PROGRAM PRG_PAOL_01_LightboxScanersCtrl
VAR

	tonEnableCameraSystem					: TON;
	bEnablePackAggregationCameraSystem		: BOOL;
	bEnablePackTriggeringAfterDelayON		: BOOL;

	tofPackAggregationCameraOFFDelay 		: TOF;
	bEnablePackTriggeringAfterDelayOFF		: BOOL;

	fbPuls							: FB_Puls;
	tonLightboxLensAirNextBlow		: TON;
	//rtLightboxLensAirBlowing		: R_TRIG;
	tonLightboxLensAirBlowing		: TOF;

	fbCameraBoxRead					: FB_2CAM_CameraBoxRead;
	aScannerCtrl					: ARRAY[1..2] OF FB_SCANNER_CameraSelect;
	aCodeDiag						: ARRAY[1..2] OF FB_SCANNER_DiagnosticLog;

	bCameraTriggersArmed			: BOOL;
	bCameraTrigger1Conditioned		: BOOL;
	bCameraTrigger2Conditioned		: BOOL;
	bCameraTrigger3Conditioned		: BOOL;
	bCameraTrigger4Conditioned		: BOOL;
	bCameraTrigger5Conditioned		: BOOL;
	bCameraTrigger6Conditioned		: BOOL;

	rtCameraTrigger					: ARRAY[0..6] OF R_TRIG;
	aCameraTrigger					: ARRAY[0..6] OF BOOL;

	fbCameraSequenceNo				: FB_2CAM_CameraSequenceNo;

	fbPackScanners_2x5Packs			: FB_2CAM_PackScanners2x5Packs;
	fbSelectCameraMap				: FB_2CAM_SelectCameraMap;

	fbAddNewOuterTriggerID			: FB_PAOL_AddNewTriggerID;
	fbMoveOuterStatusArray			: FB_PACK_MoveOuterStatusArray;	(*Actually is moving OCVPackStatusArray*)

	aAddPackCodes					: ARRAY[1..2] OF FB_2CAM_AddPackCodes;
	aPackScanner					: ARRAY[1..2] OF ST_SCANNER_CameraMap;
	aPackCameraEvaluation			: ARRAY[1..2] OF FB_SCANNER_Evaluation;

	bPackCodeDataInvalid			: BOOL;
	ctuConsecutiveDataInvalid		: CTU;

	aInfeedCamerasSync 				: ARRAY[1..2] OF FB_PAOL_InfeedCamerasSync;

	tonDelayStopOuter				: TON;


END_VAR
VAR // added by the converter: edge detectors and wires of the graphical bodies
    _w1, _w3 : BOOL;
    _w2 : UDINT;
END_VAR

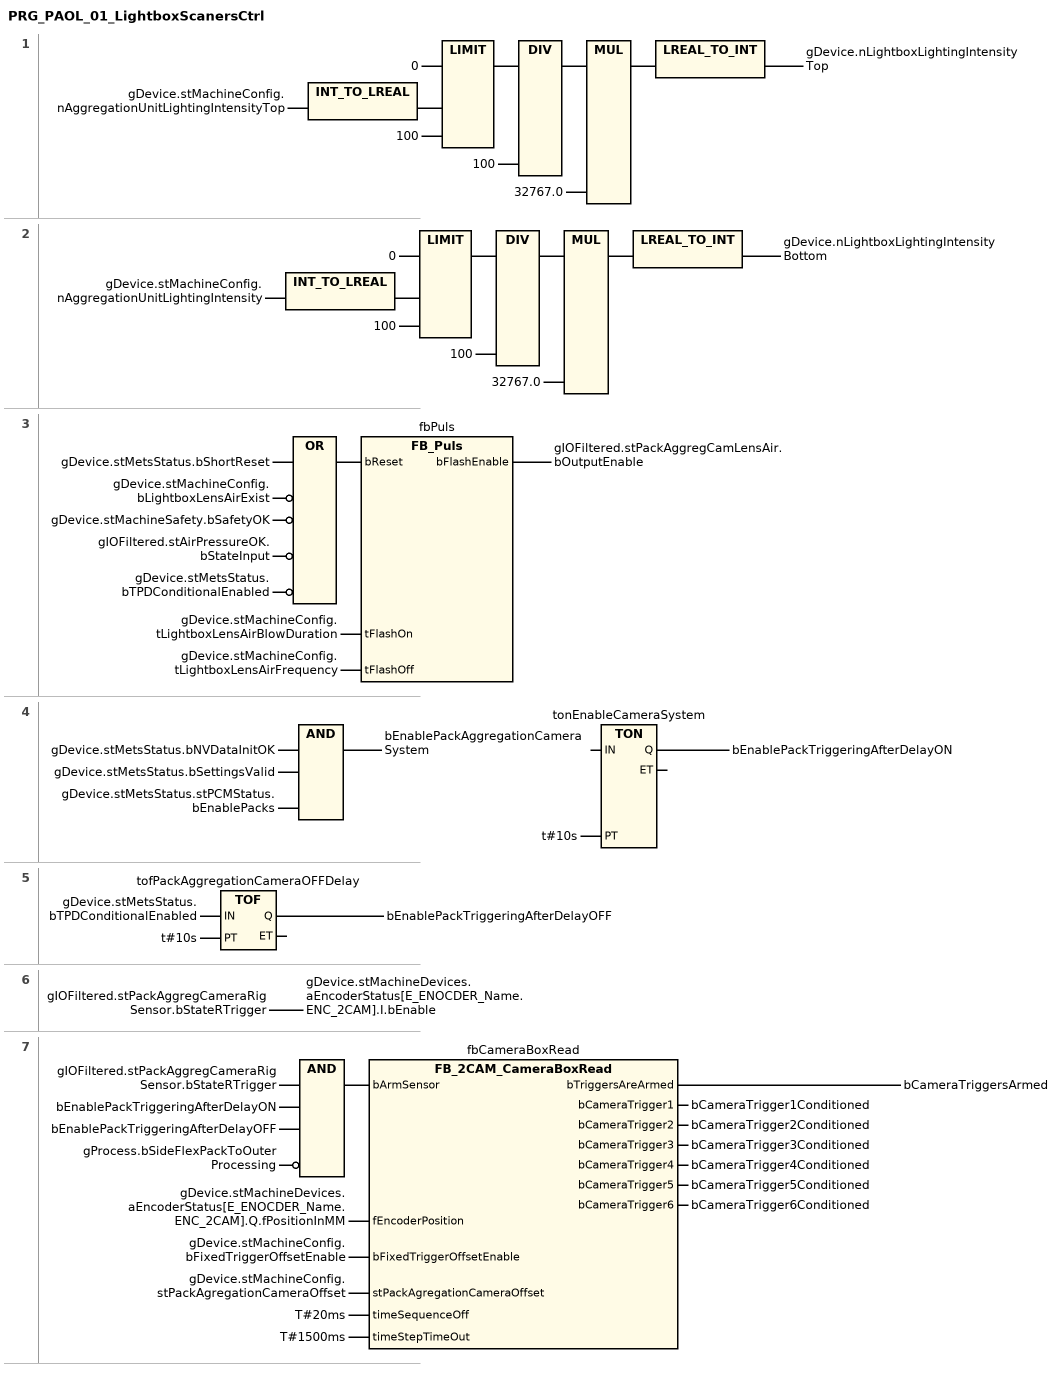
// NETWORK 1
gDevice.nLightboxLightingIntensityTop := LREAL_TO_INT((LIMIT(0, INT_TO_LREAL(gDevice.stMachineConfig.nAggregationUnitLightingIntensityTop), 100) / 100) * 32767.0);

// NETWORK 2
gDevice.nLightboxLightingIntensityBottom := LREAL_TO_INT((LIMIT(0, INT_TO_LREAL(gDevice.stMachineConfig.nAggregationUnitLightingIntensity), 100) / 100) * 32767.0);

// NETWORK 3
fbPuls(
    bReset := gDevice.stMetsStatus.bShortReset OR NOT gDevice.stMachineConfig.bLightboxLensAirExist OR NOT gDevice.stMachineSafety.bSafetyOK OR NOT gIOFiltered.stAirPressureOK.bStateInput OR NOT gDevice.stMetsStatus.bTPDConditionalEnabled,
    tFlashOn := gDevice.stMachineConfig.tLightboxLensAirBlowDuration,
    tFlashOff := gDevice.stMachineConfig.tLightboxLensAirFrequency); // FB_Puls
gIOFiltered.stPackAggregCamLensAir.bOutputEnable := fbPuls.bFlashEnable;

// NETWORK 4
_w1 := gDevice.stMetsStatus.bNVDataInitOK AND gDevice.stMetsStatus.bSettingsValid AND gDevice.stMetsStatus.stPCMStatus.bEnablePacks;
bEnablePackAggregationCameraSystem := _w1;
tonEnableCameraSystem(IN := _w1, PT := t#10s); // TON
bEnablePackTriggeringAfterDelayON := tonEnableCameraSystem.Q;

// NETWORK 5
tofPackAggregationCameraOFFDelay(IN := gDevice.stMetsStatus.bTPDConditionalEnabled, PT := t#10s); // TOF
bEnablePackTriggeringAfterDelayOFF := tofPackAggregationCameraOFFDelay.Q;

// NETWORK 6
gDevice.stMachineDevices.aEncoderStatus[E_ENOCDER_Name.ENC_2CAM].I.bEnable := gIOFiltered.stPackAggregCameraRigSensor.bStateRTrigger;

// NETWORK 7
fbCameraBoxRead(
    bArmSensor := gIOFiltered.stPackAggregCameraRigSensor.bStateRTrigger AND bEnablePackTriggeringAfterDelayON AND bEnablePackTriggeringAfterDelayOFF AND NOT gProcess.bSideFlexPackToOuterProcessing,
    fEncoderPosition := gDevice.stMachineDevices.aEncoderStatus[E_ENOCDER_Name.ENC_2CAM].Q.fPositionInMM,
    bFixedTriggerOffsetEnable := gDevice.stMachineConfig.bFixedTriggerOffsetEnable,
    stPackAgregationCameraOffset := gDevice.stMachineConfig.stPackAgregationCameraOffset,
    timeSequenceOff := T#20ms,
    timeStepTimeOut := T#1500ms,
    bCameraTrigger1 => bCameraTrigger1Conditioned,
    bCameraTrigger2 => bCameraTrigger2Conditioned,
    bCameraTrigger3 => bCameraTrigger3Conditioned,
    bCameraTrigger4 => bCameraTrigger4Conditioned,
    bCameraTrigger5 => bCameraTrigger5Conditioned,
    bCameraTrigger6 => bCameraTrigger6Conditioned); // FB_2CAM_CameraBoxRead
bCameraTriggersArmed := fbCameraBoxRead.bTriggersAreArmed;

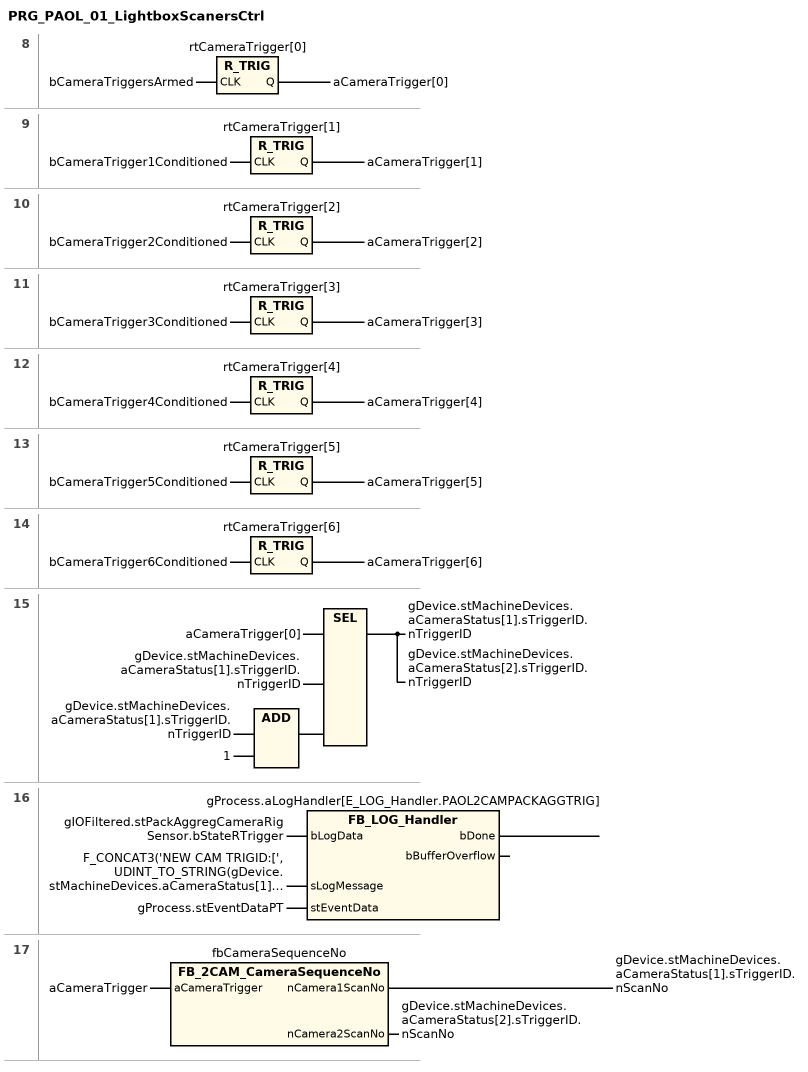
// NETWORK 8
rtCameraTrigger[0](CLK := bCameraTriggersArmed); // R_TRIG
aCameraTrigger[0] := rtCameraTrigger[0].Q;

// NETWORK 9
rtCameraTrigger[1](CLK := bCameraTrigger1Conditioned); // R_TRIG
aCameraTrigger[1] := rtCameraTrigger[1].Q;

// NETWORK 10
rtCameraTrigger[2](CLK := bCameraTrigger2Conditioned); // R_TRIG
aCameraTrigger[2] := rtCameraTrigger[2].Q;

// NETWORK 11
rtCameraTrigger[3](CLK := bCameraTrigger3Conditioned); // R_TRIG
aCameraTrigger[3] := rtCameraTrigger[3].Q;

// NETWORK 12
rtCameraTrigger[4](CLK := bCameraTrigger4Conditioned); // R_TRIG
aCameraTrigger[4] := rtCameraTrigger[4].Q;

// NETWORK 13
rtCameraTrigger[5](CLK := bCameraTrigger5Conditioned); // R_TRIG
aCameraTrigger[5] := rtCameraTrigger[5].Q;

// NETWORK 14
rtCameraTrigger[6](CLK := bCameraTrigger6Conditioned); // R_TRIG
aCameraTrigger[6] := rtCameraTrigger[6].Q;

// NETWORK 15
_w2 := SEL(aCameraTrigger[0], gDevice.stMachineDevices.aCameraStatus[1].sTriggerID.nTriggerID, gDevice.stMachineDevices.aCameraStatus[1].sTriggerID.nTriggerID + 1);
gDevice.stMachineDevices.aCameraStatus[1].sTriggerID.nTriggerID := _w2;
gDevice.stMachineDevices.aCameraStatus[2].sTriggerID.nTriggerID := _w2;

// NETWORK 16
gProcess.aLogHandler[E_LOG_Handler.PAOL2CAMPACKAGGTRIG](
    bLogData := gIOFiltered.stPackAggregCameraRigSensor.bStateRTrigger,
    sLogMessage := F_CONCAT3('NEW CAM TRIGID:[', UDINT_TO_STRING(gDevice.stMachineDevices.aCameraStatus[1].sTriggerID.nTriggerID), ']'),
    stEventData := gProcess.stEventDataPT); // FB_LOG_Handler

// NETWORK 17
fbCameraSequenceNo(aCameraTrigger := aCameraTrigger, nCamera2ScanNo => gDevice.stMachineDevices.aCameraStatus[2].sTriggerID.nScanNo); // FB_2CAM_CameraSequenceNo
gDevice.stMachineDevices.aCameraStatus[1].sTriggerID.nScanNo := fbCameraSequenceNo.nCamera1ScanNo;

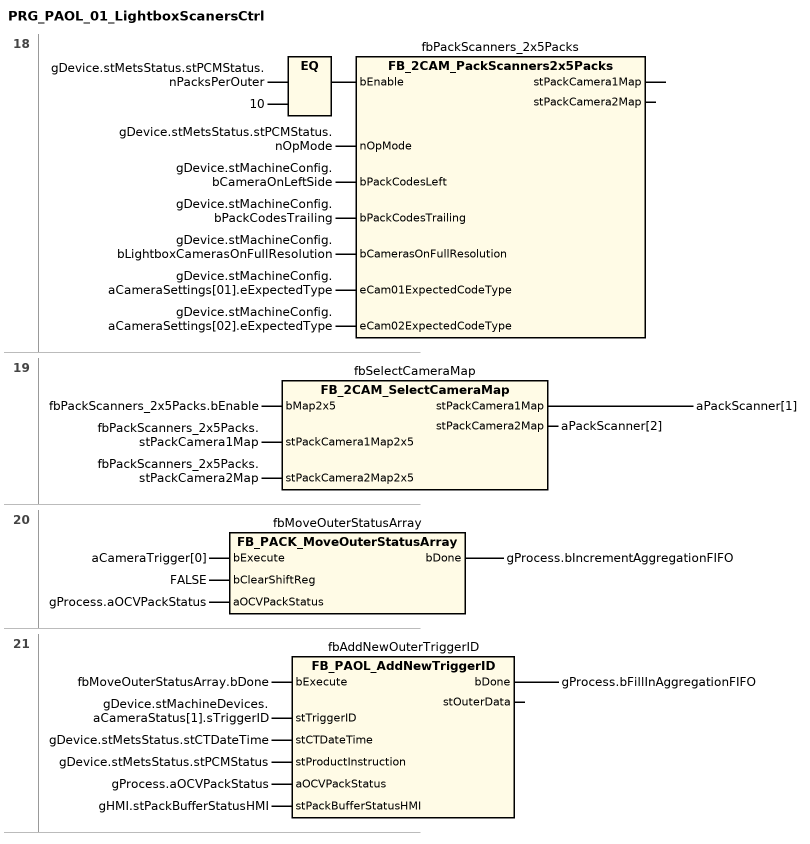
// NETWORK 18
fbPackScanners_2x5Packs(
    bEnable := gDevice.stMetsStatus.stPCMStatus.nPacksPerOuter = 10,
    nOpMode := gDevice.stMetsStatus.stPCMStatus.nOpMode,
    bPackCodesLeft := gDevice.stMachineConfig.bCameraOnLeftSide,
    bPackCodesTrailing := gDevice.stMachineConfig.bPackCodesTrailing,
    bCamerasOnFullResolution := gDevice.stMachineConfig.bLightboxCamerasOnFullResolution,
    eCam01ExpectedCodeType := gDevice.stMachineConfig.aCameraSettings[01].eExpectedType,
    eCam02ExpectedCodeType := gDevice.stMachineConfig.aCameraSettings[02].eExpectedType); // FB_2CAM_PackScanners2x5Packs

// NETWORK 19
fbSelectCameraMap(
    bMap2x5 := fbPackScanners_2x5Packs.bEnable,
    stPackCamera1Map2x5 := fbPackScanners_2x5Packs.stPackCamera1Map,
    stPackCamera2Map2x5 := fbPackScanners_2x5Packs.stPackCamera2Map,
    stPackCamera2Map => aPackScanner[2]); // FB_2CAM_SelectCameraMap
aPackScanner[1] := fbSelectCameraMap.stPackCamera1Map;

// NETWORK 20
fbMoveOuterStatusArray(
    bExecute := aCameraTrigger[0],
    bClearShiftReg := FALSE,
    aOCVPackStatus := gProcess.aOCVPackStatus); // FB_PACK_MoveOuterStatusArray
gProcess.bIncrementAggregationFIFO := fbMoveOuterStatusArray.bDone;

// NETWORK 21
fbAddNewOuterTriggerID(
    bExecute := fbMoveOuterStatusArray.bDone,
    stTriggerID := gDevice.stMachineDevices.aCameraStatus[1].sTriggerID,
    stCTDateTime := gDevice.stMetsStatus.stCTDateTime,
    stProductInstruction := gDevice.stMetsStatus.stPCMStatus,
    aOCVPackStatus := gProcess.aOCVPackStatus,
    stPackBufferStatusHMI := gHMI.stPackBufferStatusHMI); // FB_PAOL_AddNewTriggerID
gProcess.bFillInAggregationFIFO := fbAddNewOuterTriggerID.bDone;

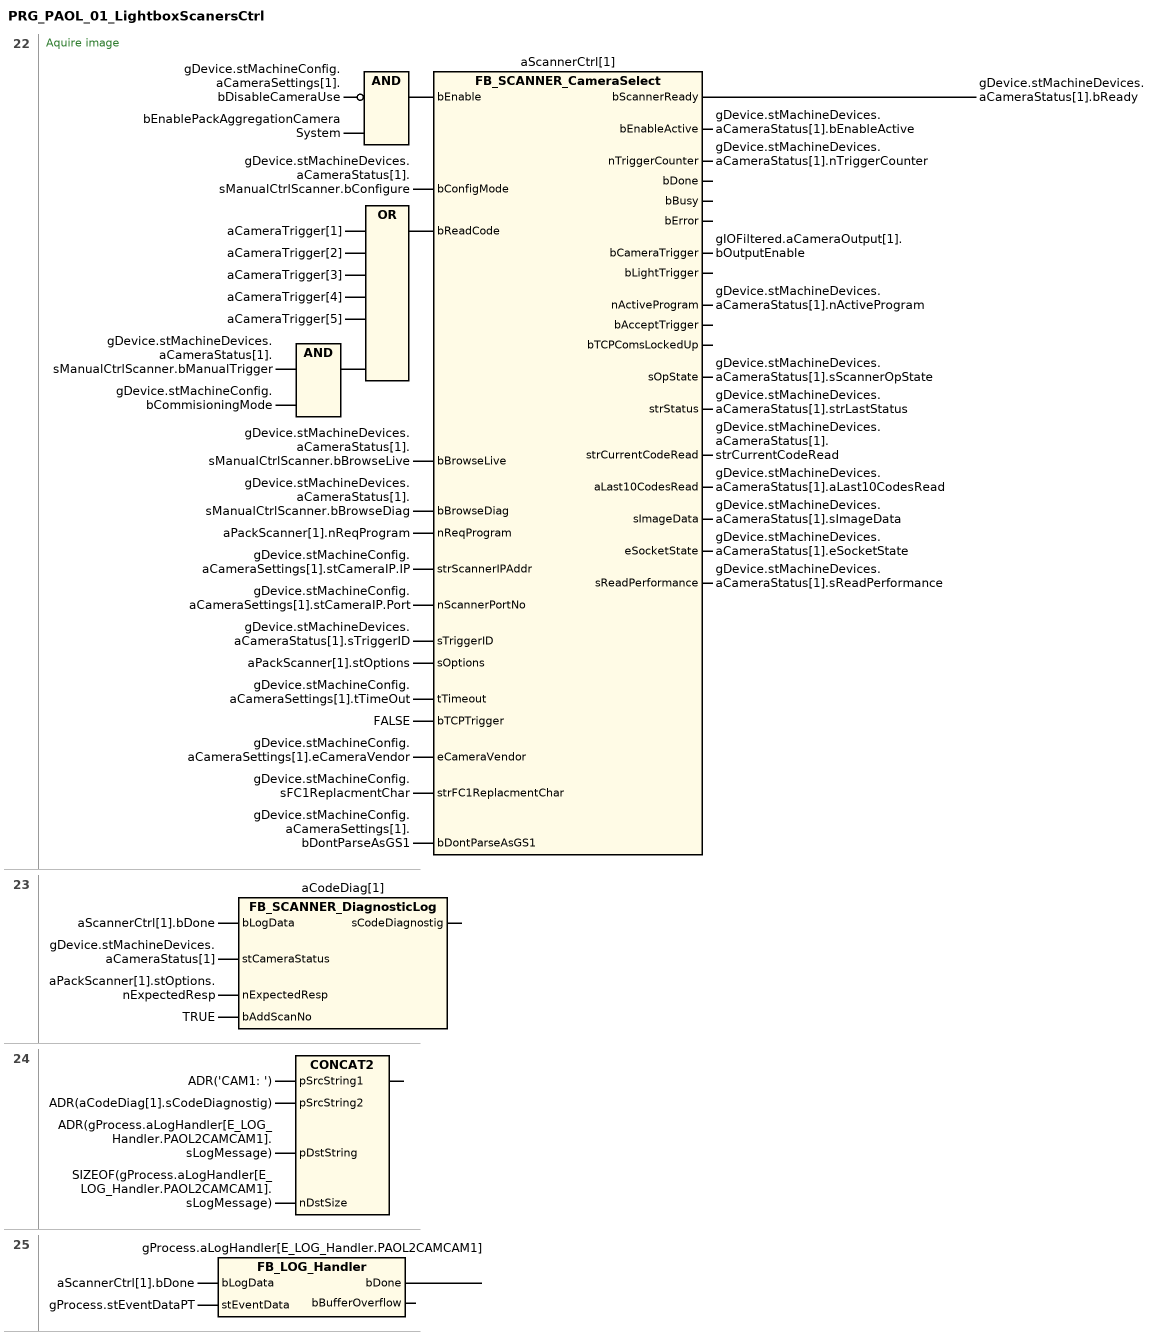
// NETWORK 22
// Aquire image
aScannerCtrl[1](
    bEnable := NOT gDevice.stMachineConfig.aCameraSettings[1].bDisableCameraUse AND bEnablePackAggregationCameraSystem,
    bConfigMode := gDevice.stMachineDevices.aCameraStatus[1].sManualCtrlScanner.bConfigure,
    bReadCode := aCameraTrigger[1] OR aCameraTrigger[2] OR aCameraTrigger[3] OR aCameraTrigger[4] OR aCameraTrigger[5] OR gDevice.stMachineDevices.aCameraStatus[1].sManualCtrlScanner.bManualTrigger AND gDevice.stMachineConfig.bCommisioningMode,
    bBrowseLive := gDevice.stMachineDevices.aCameraStatus[1].sManualCtrlScanner.bBrowseLive,
    bBrowseDiag := gDevice.stMachineDevices.aCameraStatus[1].sManualCtrlScanner.bBrowseDiag,
    nReqProgram := aPackScanner[1].nReqProgram,
    strScannerIPAddr := gDevice.stMachineConfig.aCameraSettings[1].stCameraIP.IP,
    nScannerPortNo := gDevice.stMachineConfig.aCameraSettings[1].stCameraIP.Port,
    sTriggerID := gDevice.stMachineDevices.aCameraStatus[1].sTriggerID,
    sOptions := aPackScanner[1].stOptions,
    tTimeout := gDevice.stMachineConfig.aCameraSettings[1].tTimeOut,
    bTCPTrigger := FALSE,
    eCameraVendor := gDevice.stMachineConfig.aCameraSettings[1].eCameraVendor,
    strFC1ReplacmentChar := gDevice.stMachineConfig.sFC1ReplacmentChar,
    bDontParseAsGS1 := gDevice.stMachineConfig.aCameraSettings[1].bDontParseAsGS1,
    bEnableActive => gDevice.stMachineDevices.aCameraStatus[1].bEnableActive,
    nTriggerCounter => gDevice.stMachineDevices.aCameraStatus[1].nTriggerCounter,
    bCameraTrigger => gIOFiltered.aCameraOutput[1].bOutputEnable,
    nActiveProgram => gDevice.stMachineDevices.aCameraStatus[1].nActiveProgram,
    sOpState => gDevice.stMachineDevices.aCameraStatus[1].sScannerOpState,
    strStatus => gDevice.stMachineDevices.aCameraStatus[1].strLastStatus,
    strCurrentCodeRead => gDevice.stMachineDevices.aCameraStatus[1].strCurrentCodeRead,
    aLast10CodesRead => gDevice.stMachineDevices.aCameraStatus[1].aLast10CodesRead,
    sImageData => gDevice.stMachineDevices.aCameraStatus[1].sImageData,
    eSocketState => gDevice.stMachineDevices.aCameraStatus[1].eSocketState,
    sReadPerformance => gDevice.stMachineDevices.aCameraStatus[1].sReadPerformance); // FB_SCANNER_CameraSelect
gDevice.stMachineDevices.aCameraStatus[1].bReady := aScannerCtrl[1].bScannerReady;

// NETWORK 23
aCodeDiag[1](
    bLogData := aScannerCtrl[1].bDone,
    stCameraStatus := gDevice.stMachineDevices.aCameraStatus[1],
    nExpectedResp := aPackScanner[1].stOptions.nExpectedResp,
    bAddScanNo := TRUE); // FB_SCANNER_DiagnosticLog

// NETWORK 24
CONCAT2(pSrcString1 := ADR('CAM1: '), pSrcString2 := ADR(aCodeDiag[1].sCodeDiagnostig), pDstString := ADR(gProcess.aLogHandler[E_LOG_Handler.PAOL2CAMCAM1].sLogMessage), nDstSize := SIZEOF(gProcess.aLogHandler[E_LOG_Handler.PAOL2CAMCAM1].sLogMessage));

// NETWORK 25
gProcess.aLogHandler[E_LOG_Handler.PAOL2CAMCAM1](bLogData := aScannerCtrl[1].bDone, stEventData := gProcess.stEventDataPT); // FB_LOG_Handler

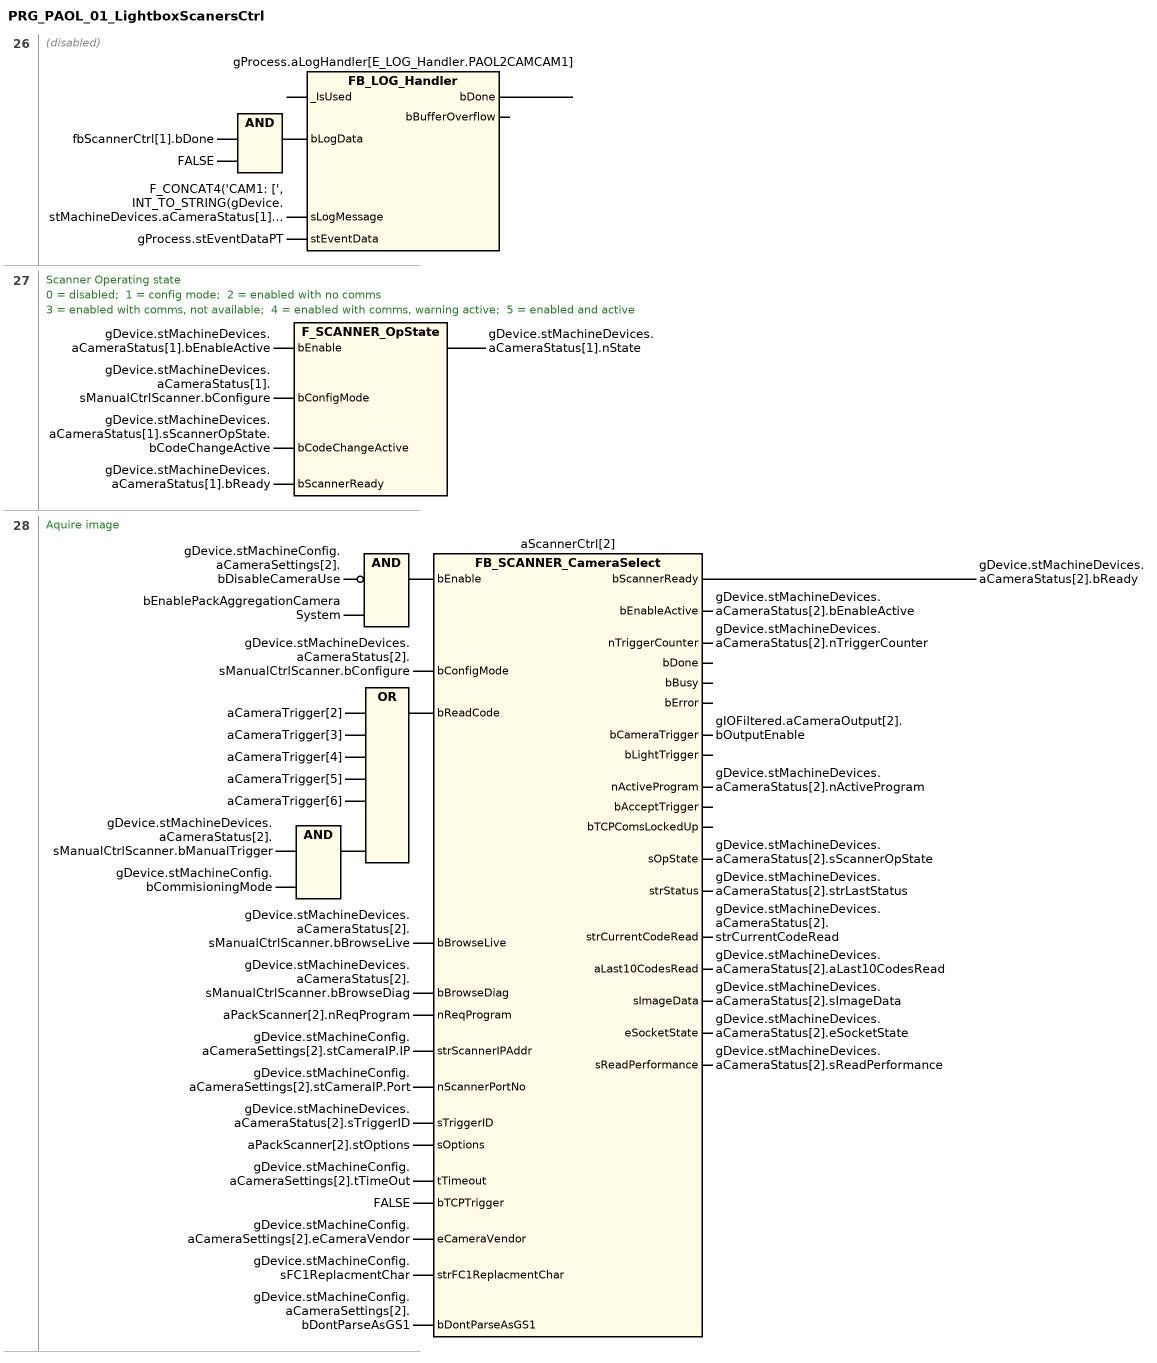
// NETWORK 26 (disabled)
// gProcess.aLogHandler[E_LOG_Handler.PAOL2CAMCAM1](
//     bLogData := fbScannerCtrl[1].bDone AND FALSE,
//     sLogMessage := F_CONCAT4('CAM1: [', INT_TO_STRING(gDevice.stMachineDevices.aCameraStatus[1].sTriggerID.nScanNo), '] - ', fbCodeDiag[1].sCodeDiagnostig),
//     stEventData := gProcess.stEventDataPT); // FB_LOG_Handler

// NETWORK 27
// 					Scanner Operating state
// 0 = disabled;  1 = config mode;  2 = enabled with no comms
// 3 = enabled with comms, not available;  4 = enabled with comms, warning active;  5 = enabled and active
//
gDevice.stMachineDevices.aCameraStatus[1].nState := F_SCANNER_OpState(bEnable := gDevice.stMachineDevices.aCameraStatus[1].bEnableActive, bConfigMode := gDevice.stMachineDevices.aCameraStatus[1].sManualCtrlScanner.bConfigure, bCodeChangeActive := gDevice.stMachineDevices.aCameraStatus[1].sScannerOpState.bCodeChangeActive, bScannerReady := gDevice.stMachineDevices.aCameraStatus[1].bReady);

// NETWORK 28
// Aquire image
aScannerCtrl[2](
    bEnable := NOT gDevice.stMachineConfig.aCameraSettings[2].bDisableCameraUse AND bEnablePackAggregationCameraSystem,
    bConfigMode := gDevice.stMachineDevices.aCameraStatus[2].sManualCtrlScanner.bConfigure,
    bReadCode := aCameraTrigger[2] OR aCameraTrigger[3] OR aCameraTrigger[4] OR aCameraTrigger[5] OR aCameraTrigger[6] OR gDevice.stMachineDevices.aCameraStatus[2].sManualCtrlScanner.bManualTrigger AND gDevice.stMachineConfig.bCommisioningMode,
    bBrowseLive := gDevice.stMachineDevices.aCameraStatus[2].sManualCtrlScanner.bBrowseLive,
    bBrowseDiag := gDevice.stMachineDevices.aCameraStatus[2].sManualCtrlScanner.bBrowseDiag,
    nReqProgram := aPackScanner[2].nReqProgram,
    strScannerIPAddr := gDevice.stMachineConfig.aCameraSettings[2].stCameraIP.IP,
    nScannerPortNo := gDevice.stMachineConfig.aCameraSettings[2].stCameraIP.Port,
    sTriggerID := gDevice.stMachineDevices.aCameraStatus[2].sTriggerID,
    sOptions := aPackScanner[2].stOptions,
    tTimeout := gDevice.stMachineConfig.aCameraSettings[2].tTimeOut,
    bTCPTrigger := FALSE,
    eCameraVendor := gDevice.stMachineConfig.aCameraSettings[2].eCameraVendor,
    strFC1ReplacmentChar := gDevice.stMachineConfig.sFC1ReplacmentChar,
    bDontParseAsGS1 := gDevice.stMachineConfig.aCameraSettings[2].bDontParseAsGS1,
    bEnableActive => gDevice.stMachineDevices.aCameraStatus[2].bEnableActive,
    nTriggerCounter => gDevice.stMachineDevices.aCameraStatus[2].nTriggerCounter,
    bCameraTrigger => gIOFiltered.aCameraOutput[2].bOutputEnable,
    nActiveProgram => gDevice.stMachineDevices.aCameraStatus[2].nActiveProgram,
    sOpState => gDevice.stMachineDevices.aCameraStatus[2].sScannerOpState,
    strStatus => gDevice.stMachineDevices.aCameraStatus[2].strLastStatus,
    strCurrentCodeRead => gDevice.stMachineDevices.aCameraStatus[2].strCurrentCodeRead,
    aLast10CodesRead => gDevice.stMachineDevices.aCameraStatus[2].aLast10CodesRead,
    sImageData => gDevice.stMachineDevices.aCameraStatus[2].sImageData,
    eSocketState => gDevice.stMachineDevices.aCameraStatus[2].eSocketState,
    sReadPerformance => gDevice.stMachineDevices.aCameraStatus[2].sReadPerformance); // FB_SCANNER_CameraSelect
gDevice.stMachineDevices.aCameraStatus[2].bReady := aScannerCtrl[2].bScannerReady;

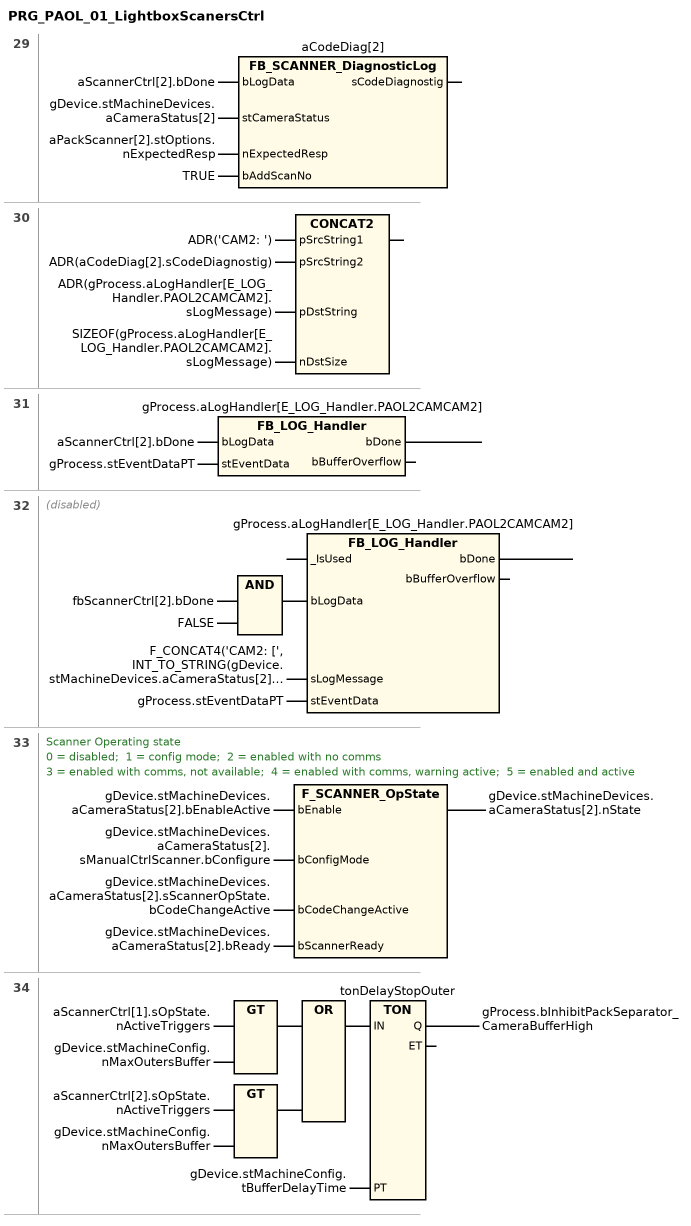
// NETWORK 29
aCodeDiag[2](
    bLogData := aScannerCtrl[2].bDone,
    stCameraStatus := gDevice.stMachineDevices.aCameraStatus[2],
    nExpectedResp := aPackScanner[2].stOptions.nExpectedResp,
    bAddScanNo := TRUE); // FB_SCANNER_DiagnosticLog

// NETWORK 30
CONCAT2(pSrcString1 := ADR('CAM2: '), pSrcString2 := ADR(aCodeDiag[2].sCodeDiagnostig), pDstString := ADR(gProcess.aLogHandler[E_LOG_Handler.PAOL2CAMCAM2].sLogMessage), nDstSize := SIZEOF(gProcess.aLogHandler[E_LOG_Handler.PAOL2CAMCAM2].sLogMessage));

// NETWORK 31
gProcess.aLogHandler[E_LOG_Handler.PAOL2CAMCAM2](bLogData := aScannerCtrl[2].bDone, stEventData := gProcess.stEventDataPT); // FB_LOG_Handler

// NETWORK 32 (disabled)
// gProcess.aLogHandler[E_LOG_Handler.PAOL2CAMCAM2](
//     bLogData := fbScannerCtrl[2].bDone AND FALSE,
//     sLogMessage := F_CONCAT4('CAM2: [', INT_TO_STRING(gDevice.stMachineDevices.aCameraStatus[2].sTriggerID.nScanNo), '] - ', fbCodeDiag[2].sCodeDiagnostig),
//     stEventData := gProcess.stEventDataPT); // FB_LOG_Handler

// NETWORK 33
// 					Scanner Operating state
// 0 = disabled;  1 = config mode;  2 = enabled with no comms
// 3 = enabled with comms, not available;  4 = enabled with comms, warning active;  5 = enabled and active
//
gDevice.stMachineDevices.aCameraStatus[2].nState := F_SCANNER_OpState(bEnable := gDevice.stMachineDevices.aCameraStatus[2].bEnableActive, bConfigMode := gDevice.stMachineDevices.aCameraStatus[2].sManualCtrlScanner.bConfigure, bCodeChangeActive := gDevice.stMachineDevices.aCameraStatus[2].sScannerOpState.bCodeChangeActive, bScannerReady := gDevice.stMachineDevices.aCameraStatus[2].bReady);

// NETWORK 34
tonDelayStopOuter(IN := aScannerCtrl[1].sOpState.nActiveTriggers > gDevice.stMachineConfig.nMaxOutersBuffer OR aScannerCtrl[2].sOpState.nActiveTriggers > gDevice.stMachineConfig.nMaxOutersBuffer, PT := gDevice.stMachineConfig.tBufferDelayTime); // TON
gProcess.bInhibitPackSeparator_CameraBufferHigh := tonDelayStopOuter.Q;

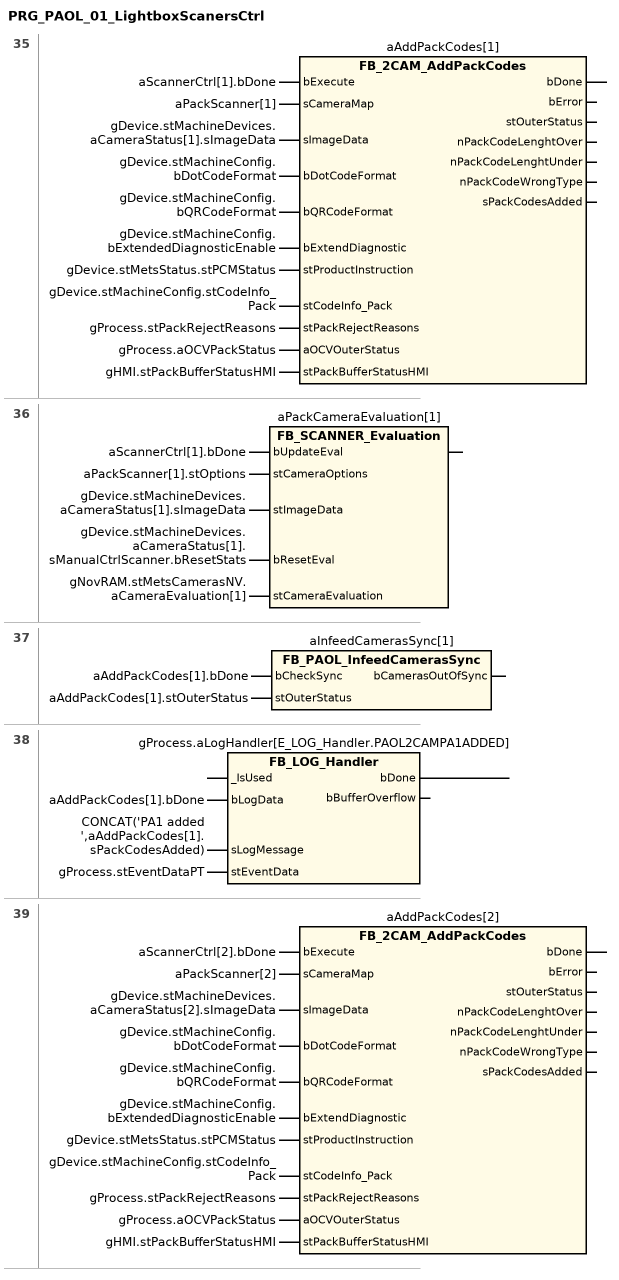
// NETWORK 35
aAddPackCodes[1](
    bExecute := aScannerCtrl[1].bDone,
    sCameraMap := aPackScanner[1],
    sImageData := gDevice.stMachineDevices.aCameraStatus[1].sImageData,
    bDotCodeFormat := gDevice.stMachineConfig.bDotCodeFormat,
    bQRCodeFormat := gDevice.stMachineConfig.bQRCodeFormat,
    bExtendDiagnostic := gDevice.stMachineConfig.bExtendedDiagnosticEnable,
    stProductInstruction := gDevice.stMetsStatus.stPCMStatus,
    stCodeInfo_Pack := gDevice.stMachineConfig.stCodeInfo_Pack,
    stPackRejectReasons := gProcess.stPackRejectReasons,
    aOCVOuterStatus := gProcess.aOCVPackStatus,
    stPackBufferStatusHMI := gHMI.stPackBufferStatusHMI); // FB_2CAM_AddPackCodes

// NETWORK 36
aPackCameraEvaluation[1](
    bUpdateEval := aScannerCtrl[1].bDone,
    stCameraOptions := aPackScanner[1].stOptions,
    stImageData := gDevice.stMachineDevices.aCameraStatus[1].sImageData,
    bResetEval := gDevice.stMachineDevices.aCameraStatus[1].sManualCtrlScanner.bResetStats,
    stCameraEvaluation := gNovRAM.stMetsCamerasNV.aCameraEvaluation[1]); // FB_SCANNER_Evaluation

// NETWORK 37
aInfeedCamerasSync[1](bCheckSync := aAddPackCodes[1].bDone, stOuterStatus := aAddPackCodes[1].stOuterStatus); // FB_PAOL_InfeedCamerasSync

// NETWORK 38
gProcess.aLogHandler[E_LOG_Handler.PAOL2CAMPA1ADDED](
    bLogData := aAddPackCodes[1].bDone,
    sLogMessage := CONCAT('PA1 added ',aAddPackCodes[1].sPackCodesAdded),
    stEventData := gProcess.stEventDataPT); // FB_LOG_Handler

// NETWORK 39
aAddPackCodes[2](
    bExecute := aScannerCtrl[2].bDone,
    sCameraMap := aPackScanner[2],
    sImageData := gDevice.stMachineDevices.aCameraStatus[2].sImageData,
    bDotCodeFormat := gDevice.stMachineConfig.bDotCodeFormat,
    bQRCodeFormat := gDevice.stMachineConfig.bQRCodeFormat,
    bExtendDiagnostic := gDevice.stMachineConfig.bExtendedDiagnosticEnable,
    stProductInstruction := gDevice.stMetsStatus.stPCMStatus,
    stCodeInfo_Pack := gDevice.stMachineConfig.stCodeInfo_Pack,
    stPackRejectReasons := gProcess.stPackRejectReasons,
    aOCVOuterStatus := gProcess.aOCVPackStatus,
    stPackBufferStatusHMI := gHMI.stPackBufferStatusHMI); // FB_2CAM_AddPackCodes

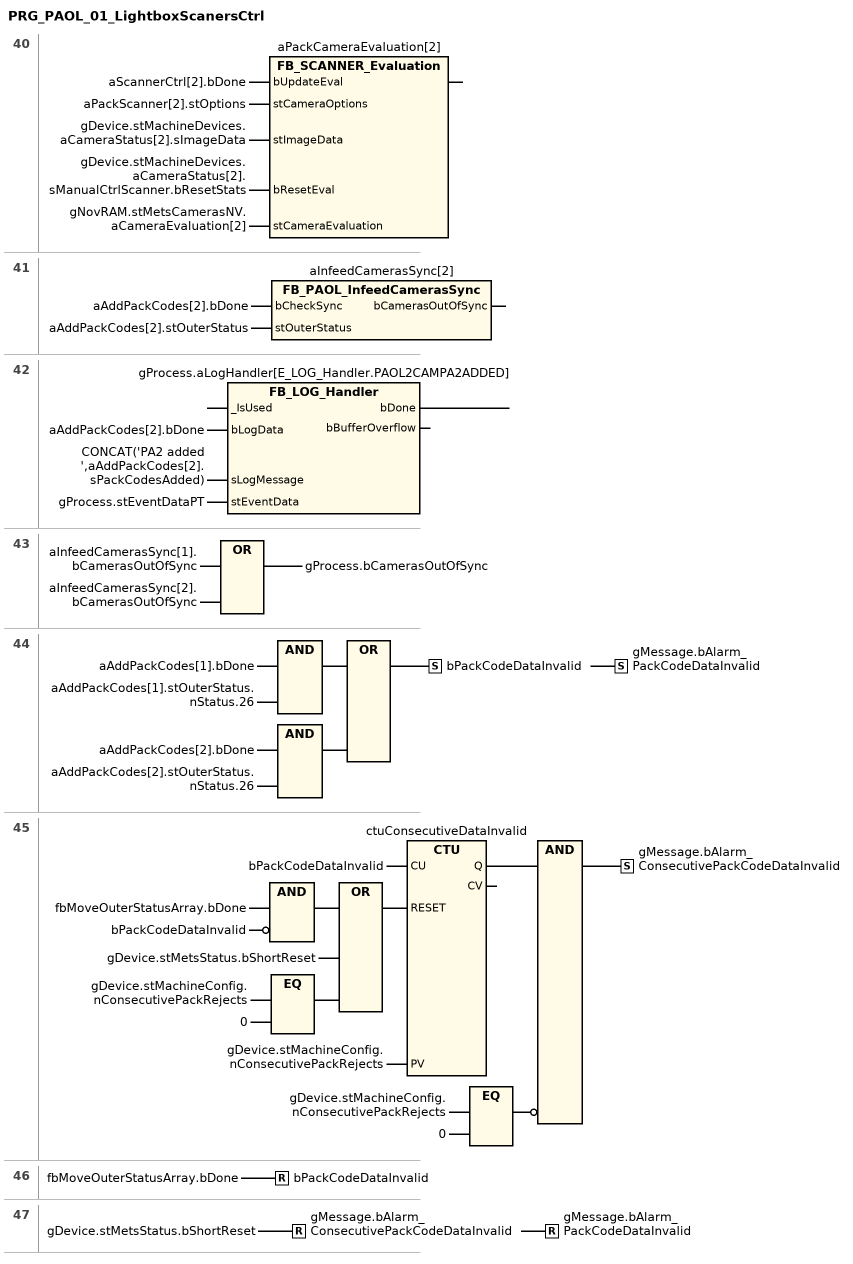
// NETWORK 40
aPackCameraEvaluation[2](
    bUpdateEval := aScannerCtrl[2].bDone,
    stCameraOptions := aPackScanner[2].stOptions,
    stImageData := gDevice.stMachineDevices.aCameraStatus[2].sImageData,
    bResetEval := gDevice.stMachineDevices.aCameraStatus[2].sManualCtrlScanner.bResetStats,
    stCameraEvaluation := gNovRAM.stMetsCamerasNV.aCameraEvaluation[2]); // FB_SCANNER_Evaluation

// NETWORK 41
aInfeedCamerasSync[2](bCheckSync := aAddPackCodes[2].bDone, stOuterStatus := aAddPackCodes[2].stOuterStatus); // FB_PAOL_InfeedCamerasSync

// NETWORK 42
gProcess.aLogHandler[E_LOG_Handler.PAOL2CAMPA2ADDED](
    bLogData := aAddPackCodes[2].bDone,
    sLogMessage := CONCAT('PA2 added ',aAddPackCodes[2].sPackCodesAdded),
    stEventData := gProcess.stEventDataPT); // FB_LOG_Handler

// NETWORK 43
gProcess.bCamerasOutOfSync := aInfeedCamerasSync[1].bCamerasOutOfSync OR aInfeedCamerasSync[2].bCamerasOutOfSync;

// NETWORK 44
_w3 := aAddPackCodes[1].bDone AND aAddPackCodes[1].stOuterStatus.nStatus.26 OR aAddPackCodes[2].bDone AND aAddPackCodes[2].stOuterStatus.nStatus.26;
bPackCodeDataInvalid S= _w3;
gMessage.bAlarm_PackCodeDataInvalid S= _w3;

// NETWORK 45
ctuConsecutiveDataInvalid(
    CU := bPackCodeDataInvalid,
    RESET := fbMoveOuterStatusArray.bDone AND NOT bPackCodeDataInvalid OR gDevice.stMetsStatus.bShortReset OR gDevice.stMachineConfig.nConsecutivePackRejects = 0,
    PV := gDevice.stMachineConfig.nConsecutivePackRejects); // CTU
gMessage.bAlarm_ConsecutivePackCodeDataInvalid S= ctuConsecutiveDataInvalid.Q AND NOT (gDevice.stMachineConfig.nConsecutivePackRejects = 0);

// NETWORK 46
bPackCodeDataInvalid R= fbMoveOuterStatusArray.bDone;

// NETWORK 47
gMessage.bAlarm_ConsecutivePackCodeDataInvalid R= gDevice.stMetsStatus.bShortReset;
gMessage.bAlarm_PackCodeDataInvalid R= gDevice.stMetsStatus.bShortReset;

END_PROGRAM

(* stored: Version 1.1.0.1
   POU PRG_PAOL_01_LightboxScanersCtrl: Id {6a599ab9-38ba-470e-b55d-231d7d6f3142}, SpecialFunc None *)
